Staubli VAL3: Tool.dtx

bool bExit
bool bListRefresh
bool bUserRefresh
mdesc mNomSpeed
num nSelected
num nType = 1
string sItem = "tool1"
string sList[20]
  [0] = "tool1"
  [1] = "tool2"
  [2] = "tool3"
  [3] = "tool4"
  [4] = "tool5"
  [5] = "tool6"
  [6] = "tool7"
  [7] = "tool8"
  [8] = "tool9"
  [9] = "tool10"
  [10] = "tool11"
  [11] = "tool12"
  [12] = "tool13"
  [13] = "tool14"
  [14] = "tool15"
  [15] = "tool16"
  [16] = "tool17"
  [17] = "tool18"
  [18] = "tool19"
  [19] = "tool20"
string sListItemValue[6]
  [0] = "0    "
  [1] = "0    "
  [2] = "100    "
  [3] = "0    "
  [4] = "0    "
  [5] = "0    "
string sParameter[6]
  [0] = "X        :0        "
  [1] = "Y        :0         "
  [2] = "Z        :100      "
  [3] = "Rx       :0         "
  [4] = "Ry       :0         "
  [5] = "Rz       :0         "
string sToolName
public tool tTool{}
  [tool1] = {z=100, fatherId=flange[0], ioLink=valve1}
  [tool10] = {fatherId=flange[0], ioLink=valve1}
  [tool11] = {fatherId=flange[0], ioLink=valve1}
  [tool12] = {fatherId=flange[0], ioLink=valve1}
  [tool13] = {fatherId=flange[0], ioLink=valve1}
  [tool14] = {fatherId=flange[0], ioLink=valve1}
  [tool15] = {fatherId=flange[0], ioLink=valve1}
  [tool16] = {fatherId=flange[0], ioLink=valve1}
  [tool17] = {fatherId=flange[0], ioLink=valve1}
  [tool18] = {fatherId=flange[0], ioLink=valve1}
  [tool19] = {fatherId=flange[0], ioLink=valve1}
  [tool2] = {fatherId=flange[0], ioLink=valve1}
  [tool20] = {fatherId=flange[0], ioLink=valve1}
  [tool3] = {fatherId=flange[0], ioLink=valve1}
  [tool4] = {fatherId=flange[0], ioLink=valve1}
  [tool5] = {fatherId=flange[0], ioLink=valve1}
  [tool6] = {fatherId=flange[0], ioLink=valve1}
  [tool7] = {fatherId=flange[0], ioLink=valve1}
  [tool8] = {fatherId=flange[0], ioLink=valve1}
  [tool9] = {fatherId=flange[0], ioLink=valve1}
